FUNCTION_BLOCK ILOCK_SR_AX (* Realizes a chainable momentary latch with interlock (AX/AX2 interface) *)
  (* Standard: 61499-1; Description: Copyright (c) 2026 Meisterschulen am Ostbahnhof *)
  (* Version 1.0, 2026-05-07, Gemini CLI, Meisterschulen am Ostbahnhof, initial version *)
  PACKAGE logiBUS::signalprocessing::interlock;
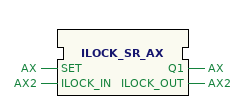
  SOCKETS
    SET : adapter::types::unidirectional::AX; (* Momentary Set signal *)
    ILOCK_IN : adapter::types::bidirectional::AX2; (* Interlock from above *)
  END_SOCKETS
  PLUGS
    Q1 : adapter::types::unidirectional::AX; (* Output *)
    ILOCK_OUT : adapter::types::bidirectional::AX2; (* Interlock to below *)
  END_PLUGS
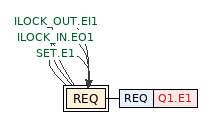
  EC_STATES
    REQ : REQ -> Q1.E1;
  END_STATES
  EC_TRANSITIONS
    REQ TO REQ := SET.E1;
    REQ TO REQ := ILOCK_IN.EO1;
    REQ TO REQ := ILOCK_OUT.EI1;
  END_TRANSITIONS
  ALGORITHM REQ IN ST:
(* Momentary latch: Q1 is active if SET is active AND no other element is set *)
Q1.D1 := SET.D1 AND NOT (ILOCK_IN.DO1 OR ILOCK_OUT.DI1);

(* Propagate status *)
ILOCK_IN.DI1 := Q1.D1;
ILOCK_OUT.DO1 := Q1.D1;
  END_ALGORITHM
END_FUNCTION_BLOCK
